PROGRAM PRG_ILK
VAR
END_VAR

(*Evaluate Global Interlocks*)

US_Roughing_Valves_Open := (fb_AT1K0_GAS_VRC_50.M_IsOpen() AND fb_AT1K0_GAS_VRC_60.M_IsOpen());
DS_Roughing_Valves_Open := (fb_AT1K0_GAS_VRC_90.M_IsOpen() AND( fb_AT1K0_GAS_PMF_90.stPump.eState = pumpRUNNING)) OR   (fb_AT1K0_GAS_VRC_100.iq_stValve.i_xOpnLS AND (fb_AT1K0_GAS_PMF_100.stPump.eState = pumpRUNNING ));
US_Turbo_Valves_Open := fb_AT1K0_GAS_VRC_10.M_IsOpen() AND  fb_AT1K0_GAS_VRC_20.M_IsOpen() AND fb_AT1K0_GAS_VRC_30.M_IsOpen() AND fb_AT1K0_GAS_VRC_40.M_IsOpen();
DS_Turbo_Valves_Open := fb_AT1K0_GAS_VRC_110.M_IsOpen() AND  fb_AT1K0_GAS_VRC_120.M_IsOpen() AND fb_AT1K0_GAS_VRC_130.M_IsOpen()AND fb_AT1K0_GAS_VRC_140.M_IsOpen();
US_Turbo_Running := (fb_AT1K0_GAS_PTM_10.iq_stPtm.eState = pumpRUNNING) AND (fb_AT1K0_GAS_PTM_20.iq_stPtm.eState = pumpRUNNING) AND (fb_AT1K0_GAS_PTM_30.iq_stPtm.eState = pumpRUNNING) AND (fb_AT1K0_GAS_PTM_40.iq_stPtm.eState = pumpRUNNING);
DS_Turbo_Running := (fb_AT1K0_GAS_PTM_110.iq_stPtm.eState = pumpRUNNING) AND (fb_AT1K0_GAS_PTM_120.iq_stPtm.eState = pumpRUNNING) AND (fb_AT1K0_GAS_PTM_130.iq_stPtm.eState = pumpRUNNING) AND (fb_AT1K0_GAS_PTM_140.iq_stPtm.eState = pumpRUNNING);

(* Link The correct override bit to the correct vacuum section*)



(*P/MPS FF*)

END_PROGRAM

(* stored: Version 1.1.0.1, ProductVersion 3.1.4022.18
   POU PRG_ILK: Id {01cec7ee-0a1e-4d0a-98ae-432579a5cf6a}, SpecialFunc None *)
